(* PLC project EP1, Desconocido Sin nombre 1 *)
(* stored: creationDateTime 2024-11-27T17:44:38, modificationDateTime 2024-11-27T18:04:00 *)

PROGRAM EP1
  VAR
    Start1 : BOOL;
    Stop1 : BOOL;
    Motor1 : BOOL;
    Start2 : BOOL;
    Stop2 : BOOL;
    Motor2 : BOOL;
    L1 : BOOL;
    L2 : BOOL;
  END_VAR

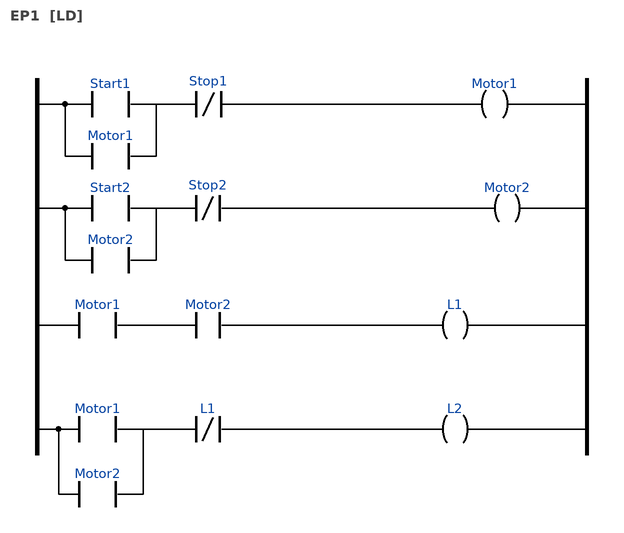
(* LD diagram, written out as Structured Text *)
Motor1 := (Start1 OR Motor1) AND NOT Stop1;
Motor2 := (Start2 OR Motor2) AND NOT Stop2;
L1 := Motor1 AND Motor2;
L2 := (Motor1 OR Motor2) AND NOT L1;
END_PROGRAM

CONFIGURATION Config0
  RESOURCE Res0 ON PLC
    TASK task0(INTERVAL := T#20ms, PRIORITY := 0);
    PROGRAM instance0 WITH task0 : EP1;
  END_RESOURCE
END_CONFIGURATION
